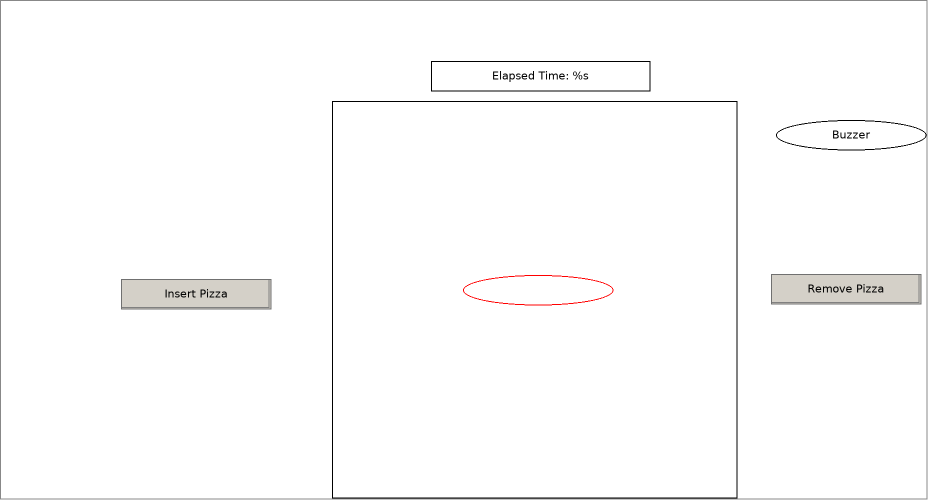
VISUALIZATION Visualization  // 928x500
    Rectangle (332,101 405x397)
    Button (121,279 150x30), "Insert Pizza"
        OnMouseDown: execute { MAIN.bPizzaInOven := TRUE; }
    Button (771,274 150x30), "Remove Pizza"
        OnMouseDown: execute { MAIN.bPizzaInOven := FALSE; }
    Ellipse (463,275 150x30), invisible if: NOT MAIN.bPizzaInOven
    Rectangle (431,61 219x30), "Elapsed Time: %s", text variable: MAIN.fbMyTimer.ET
    Ellipse (776,120 150x30), "Buzzer", colour toggle: MAIN.bBuzzer
END_VISUALIZATION

(* stored: Version 1.1.0.1, ProductVersion 3.1.4019.2
   Visu Visualization: Id {41ffcbcf-8956-4c45-9483-1f86be3ae1ed} *)
